FUNCTION_BLOCK S_TO_S (* Tamplate for a simple Basic Function Block Type *)
  (* Standard: 61499-2 *)
  (* Version 0.0, 2018-07-30, 4DIAC-IDE, 4DIAC-Consortium *)
  (* Version 1.0, 2016-05-26, AZ, fortiss GmbH *)
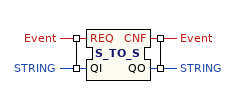
  EVENT_INPUT
    REQ WITH QI; (* Normal Execution Request *)
  END_EVENT
  EVENT_OUTPUT
    CNF WITH QO; (* Execution Confirmation *)
  END_EVENT
  VAR_INPUT
    QI : STRING; (* Input event qualifier *)
  END_VAR
  VAR_OUTPUT
    QO : STRING; (* Output event qualifier *)
  END_VAR
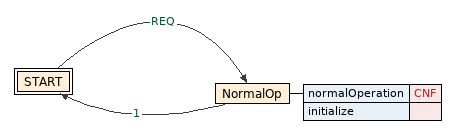
  EC_STATES
    START; (* Initial State *)
    NormalOp : normalOperation -> CNF, initialize; (* Normal execution *)
  END_STATES
  EC_TRANSITIONS
    START TO NormalOp := REQ;
    NormalOp TO START := 1;
  END_TRANSITIONS
  ALGORITHM initialize IN ST: (* Initialization algorithm *)
QO := "";
  END_ALGORITHM
  ALGORITHM normalOperation IN ST: (* new algorithm *)
QO := QI;
  END_ALGORITHM
END_FUNCTION_BLOCK
